FUNCTION_BLOCK fbInheritanceLevel_2 EXTENDS fbInheritanceLevel_1
VAR
	{attribute addProperty Name "LEVEL 2"}
	level_2 : stAllTypes;
END_VAR

SUPER^();

METHOD Init : BOOL
VAR_INPUT
END_VAR
SUPER^.Init();
END_METHOD

END_FUNCTION_BLOCK

(* stored: Version 1.1.0.1, ProductVersion 3.1.4022.12
   POU fbInheritanceLevel_2: Id {59454bff-4d66-4402-b31c-ed00b6954983}, SpecialFunc None
   Method Init: Id {32feb95a-c3f5-4923-8c40-01d1fbb81388} *)
